TYPE DUT_Position :
STRUCT
	x					: LREAL;
	y					: LREAL;
	z					: LREAL;
	a					: LREAL;
	b					: LREAL;
	c					: LREAL;
END_STRUCT
END_TYPE

(* stored: Version 1.1.0.1, ProductVersion 3.1.4024.12
   DUT DUT_Position: Id {5844358f-de1c-4b98-83f8-cc1b677e6160} *)
